# B&R Automation Studio project Palletizer (part 2)

#### Crane.st - Cyclic code
```iecst
PROGRAM _CYCLIC

	CASE State OF

		C_StopSequence:

			StartCrane			:= FALSE;
			GantryCrane.Command	:= EMERGENCY_STOP_REQUEST;
			BoxCrane.Command	:= EMERGENCY_STOP_REQUEST;
			State				:= C_StopDONE;

		C_StopDONE:

			IF (GantryCranePositionReached AND BoxCranePositionReached) THEN
				GantryCrane.Command	 := IDLE;
				BoxCrane.Command	 := IDLE;
				Crane_EmergencyStop  := FALSE;
				Crane_ImmediateStop  := FALSE;
				Crane_OnPhaseStop	 := FALSE;
				StopRequest			 := TRUE;
				State				 := C_WaitStart;
			END_IF;

		C_ResetConfig:

			IF NOT Crane_ResetConfig THEN
				State	:= C_WaitStart;
			END_IF;

			IF (GantryCranePositionReached AND BoxCranePositionReached AND NOT SlideRail_disable_request
				AND NOT PusherZ_enable_request AND NOT PusherX_enable_request AND NOT Vacuum_disable_request
				AND NOT Cartboard_disable_request) THEN

				GantryCrane.Command	:= IDLE;
				BoxCrane.Command	:= IDLE;

				FOR i := 0 TO 9 DO
					GD_StatusRequest[i]	:= FALSE;
				END_FOR;

				Crane_ResetConfig := FALSE;
				State			  := C_WaitStart;

			END_IF;

		C_RestoreConfig1:

			GantryCrane.Command	:= IDLE;
			BoxCrane.Command	:= IDLE;

			FOR i := 0 TO 9 DO
				IF GD_StatusRequest[i] THEN
					CASE i OF
						0:	Vacuum_enable_request	  := TRUE;
						1:	Vacuum_disable_request	  := TRUE;
						2:	Cartboard_enable_request  := TRUE;
						3:	Cartboard_disable_request := TRUE;
						4:	SlideRail_enable_request  := TRUE;
						5:	SlideRail_disable_request := TRUE;
						6:	PusherZ_enable_request	  := TRUE;
						7:	PusherZ_disable_request	  := TRUE;
						8:	PusherX_enable_request	  := TRUE;
						9:	PusherX_disable_request	  := TRUE;
					END_CASE;
				END_IF;
			END_FOR;

			Enable_Disable_Counter	:= 70;
			State					:= C_RestoreConfig2;

		C_RestoreConfig2:

			FOR i := 0 TO 9 DO
				IF GD_StatusRequest[i] THEN
					CASE i OF

						0:  IF NOT Vacuum_enable_request THEN
								GD_StatusRequest[i]	:= FALSE;
							END_IF;

						1:  IF NOT Vacuum_disable_request THEN
								GD_StatusRequest[i]	:= FALSE;
							END_IF;

						2:  IF NOT Cartboard_enable_request THEN
								GD_StatusRequest[i]	:= FALSE;
							END_IF

						3:  IF NOT Cartboard_disable_request THEN
								GD_StatusRequest[i]	:= FALSE;
							END_IF;

						4:	IF NOT SlideRail_enable_request THEN
								GD_StatusRequest[i]	:= FALSE;
							END_IF;

						5:  IF NOT SlideRail_disable_request THEN
								GD_StatusRequest[i]	:= FALSE;
							END_IF;

						6:  IF NOT PusherZ_enable_request THEN
								GD_StatusRequest[i]	:= FALSE;
							END_IF;

						7:  IF NOT PusherZ_disable_request THEN
								GD_StatusRequest[i]	:= FALSE;
							END_IF;

						8:  IF NOT PusherX_enable_request THEN
								GD_StatusRequest[i]	:= FALSE;
							END_IF;

						9:  IF NOT PusherX_disable_request THEN
								GD_StatusRequest[i]	:= FALSE;
							END_IF;

					END_CASE;
				END_IF;
			END_FOR;

			Enable_Disable_Counter	:= Enable_Disable_Counter - 1;

			IF Enable_Disable_Counter = 0 THEN

				IF CheckPosition[0] THEN
					GantryCraneSetPoint	:= OldPosition[0];
					GantryCrane.Command	:= CHANGE_POSITION;
				END_IF;

				IF CheckPosition[1] THEN
					BoxCraneSetPoint	:= OldPosition[1];
					BoxCrane.Command	:= CHANGE_POSITION;
				END_IF;

				State	:= C_RestoreConfig3;
			END_IF;

		C_RestoreConfig3:

			IF (GantryCranePositionReached AND CheckPosition[0]) THEN
				GantryCranePositionRestored	:= TRUE;
				GantryCrane.Command			:= IDLE;
			END_IF;

			IF (BoxCranePositionReached AND CheckPosition[1]) THEN
				BoxCranePositionRestored := TRUE;
				BoxCrane.Command		 := IDLE;
			END_IF;

			IF (NOT CheckPosition[0] OR GantryCranePositionRestored) AND (NOT CheckPosition[1] OR BoxCranePositionRestored) THEN
				StopRequest	   := FALSE;
				Crane_Restart  := FALSE;
				State		   := OldState;
			END_IF;

		C_WaitStart:

			IF Crane_Restart THEN
	  			State := C_RestoreConfig1;
			END_IF;

			IF Crane_ResetConfig THEN
				CraneCartboardCounter	  := 28;
				CraneReady				  := FALSE;
				HoldBoxes				  := FALSE;
				LoadBoxesOnPallet		  := FALSE;
				BoxesOnPallet			  := FALSE;
				SlideRail_disable_request := TRUE;
				PusherZ_enable_request	  := TRUE; (* pusher down *)
				PusherX_enable_request	  := TRUE; (* pusher forward *)
				Vacuum_disable_request	  := TRUE;
				Cartboard_disable_request := TRUE;
				GantryCraneSetPoint		  := 0;
				GantryCrane.Command	      := CHANGE_POSITION;
				BoxCraneSetPoint	      := 0;
				BoxCrane.Command	      := CHANGE_POSITION;
				State	                  := C_ResetConfig;
			END_IF;

			IF (StartCrane AND NOT Crane_ResetConfig AND NOT Crane_Restart) THEN
				GantryCraneSetPoint	 := 0;
				GantryCrane.Command	 := CHANGE_POSITION;
				State				 := C_WaitGantryCraneStartPosition;
			END_IF;

			IF Crane_EmergencyStop THEN
				State	:= C_StopSequence;
			END_IF;

			IF Crane_ImmediateStop AND NOT StopRequest THEN
				OldState := State;
				State	 := C_StopSequence;
			END_IF;

			IF Crane_ImmediateStop AND StopRequest THEN
				State	:= C_StopSequence;
			END_IF;

		C_WaitGantryCraneStartPosition:

			IF (GantryCranePositionReached OR GantryCranePositionRestored) THEN
				CheckPosition[0]			:= FALSE;
				GantryCranePositionRestored	:= FALSE;
				GantryCrane.Command			:= IDLE;
				BoxCraneSetPoint			:= -0.195;
				BoxCrane.Command			:= CHANGE_POSITION;
				State						:= C_WaitCartboardLoadPosition;
			END_IF;

			IF Crane_EmergencyStop THEN
				State	:= C_StopSequence;
			END_IF;

			IF Crane_ImmediateStop THEN
				CheckPosition[0] := TRUE;
				OldPosition[0]	 := 0;  (* old Gantry Position *)
				OldState		 := State;
				State			 := C_StopSequence;
			END_IF;

		C_WaitCartboardLoadPosition:

			IF (BoxCranePositionReached OR BoxCranePositionRestored) THEN
				CheckPosition[1]		 := FALSE;
				BoxCranePositionRestored := FALSE;
				BoxCrane.Command		 := IDLE;
				Vacuum_enable_request	 := TRUE;
				Cartboard_enable_request := TRUE;
				State					 := C_WaitCartboardLoad;
			END_IF;

			IF Crane_EmergencyStop THEN
				State	:= C_StopSequence;
			END_IF;

			IF Crane_ImmediateStop THEN
				CheckPosition[1] := TRUE;
				OldPosition[1]	 := -0.195;  (* old Box Position *)
				OldState		 := State;
				State			 := C_StopSequence;
			END_IF;

		C_WaitCartboardLoad:

			IF (NOT Vacuum_enable_request AND NOT Cartboard_enable_request) THEN
				BoxCraneSetPoint	:= 0;
				BoxCrane.Command	:= CHANGE_POSITION;
	  			State				:= C_WaitBoxCraneStartPosition;
			END_IF;

			IF Crane_EmergencyStop THEN
				State := C_StopSequence;
			END_IF;

			IF Crane_ImmediateStop THEN
				GD_StatusRequest[0] := TRUE; (* vacuumEN *)
				GD_StatusRequest[2] := TRUE; (* cartboardEN *)
				OldState		    := State;
				State				:= C_StopSequence;
			END_IF;

		C_WaitBoxCraneStartPosition:

			IF (BoxCranePositionReached OR BoxCranePositionRestored)THEN
				CheckPosition[1]		 := FALSE;
				BoxCranePositionRestored := FALSE;
				BoxCrane.Command		 := IDLE;
				PusherZ_enable_request 	 := TRUE; (* pusher down *)
				State					 := C_WaitPusherZStartDown;
			END_IF;

			IF Crane_EmergencyStop THEN
				State	:= C_StopSequence;
			END_IF;

			IF Crane_ImmediateStop THEN
				CheckPosition[1] := TRUE;
				OldPosition[1]	 := 0;  (* old Box Position *)
				OldState		 := State;
				State			 := C_StopSequence;
			END_IF;

		C_WaitPusherZStartDown:

			IF NOT PusherZ_enable_request THEN
				PusherX_enable_request := TRUE; (* pusher forward *)
				State				   := C_WaitPusherXStartFwd;
			END_IF;

			IF Crane_EmergencyStop THEN
				State	:= C_StopSequence;
			END_IF;

			IF Crane_ImmediateStop THEN
				GD_StatusRequest[6] := TRUE; (* PusherZ_EN *)
				OldState			:= State;
				State				:= C_StopSequence;
			END_IF;

		C_WaitPusherXStartFwd:

			IF NOT PusherX_enable_request THEN
				Cartboard_disable_request := TRUE;
				State					  := C_LockCartboard;
			END_IF;

			IF Crane_EmergencyStop THEN
				State	:= C_StopSequence;
			END_IF;

			IF Crane_ImmediateStop THEN
				GD_StatusRequest[8] := TRUE; (* PusherX_EN *)
				OldState		    := State;
				State				:= C_StopSequence;
			END_IF;

		C_LockCartboard:

			IF NOT Cartboard_disable_request THEN
				CraneCartboardCounter	:= CraneCartboardCounter - 1;
				CraneReady				:= TRUE;
				State					:= C_WaitBoxes;
			END_IF;

			IF Crane_EmergencyStop THEN
				State	:= C_StopSequence;
			END_IF;

			IF Crane_ImmediateStop THEN
				GD_StatusRequest[3] := TRUE; (* CartboardDIS *)
				OldState			:= State;
				State				:= C_StopSequence;
			END_IF;

		C_WaitBoxes:

			IF HoldBoxes THEN
				SlideRail_enable_request := TRUE;
				State					 := C_WaitSlideRailHold;
			END_IF;

			IF Crane_EmergencyStop THEN
				State	:= C_StopSequence;
			END_IF;

			IF Crane_ImmediateStop OR Crane_OnPhaseStop THEN
				OldState := State;
				State	 := C_StopSequence;
			END_IF;

		C_WaitSlideRailHold:

			IF NOT SlideRail_enable_request THEN
				PusherZ_disable_request	:= TRUE; (* pusher up *)
				State					:= C_WaitPusherZPushUp;
			END_IF;

			IF Crane_EmergencyStop THEN
				State	:= C_StopSequence;
			END_IF;

			IF Crane_ImmediateStop THEN
				GD_StatusRequest[4] := TRUE; (* SlideRailEN *)
				OldState			:= State;
				State				:= C_StopSequence;
			END_IF;

		C_WaitPusherZPushUp:

			IF NOT PusherZ_disable_request THEN
				PusherX_disable_request	:= TRUE; (* pusher backward *)
				State					:= C_WaitPusherXPushBwd;
			END_IF;

			IF Crane_EmergencyStop THEN
				State	:= C_StopSequence;
			END_IF;

			IF Crane_ImmediateStop THEN
				GD_StatusRequest[7] := TRUE; (* PusherZ_DIS *)
				OldState			:= State;
				State				:= C_StopSequence;
			END_IF;

		C_WaitPusherXPushBwd:

			IF NOT PusherX_disable_request THEN
				PusherZ_enable_request := TRUE; (* pusher down *)
	  			State				   := C_Idle;
			END_IF;

			IF Crane_EmergencyStop THEN
				State	:= C_StopSequence;
			END_IF;

			IF Crane_ImmediateStop THEN
				GD_StatusRequest[9] := TRUE; (* PusherX_DIS *)
				OldState			:= State;
				State				:= C_StopSequence;
			END_IF;

		C_Idle:

			IF (LoadBoxesOnPallet AND NOT PusherZ_enable_request) THEN
	  			State	:= C_WaitPusherZPushDown;
			END_IF;

			IF Crane_EmergencyStop THEN
				State	:= C_StopSequence;
			END_IF;

			IF Crane_ImmediateStop THEN
				GD_StatusRequest[6] := TRUE; (* PusherZ_EN *)
				OldState		    := State;
				State				:= C_StopSequence;
			END_IF;

		C_WaitPusherZPushDown:

			IF NOT SecondLayer THEN
				BoxCraneSetPoint := -0.2;
				BoxCrane.Command := CHANGE_POSITION;
				State			 := C_WaitBoxCraneCartboardPos;
			END_IF;

			IF SecondLayer THEN
				BoxCraneSetPoint := 0.01;
				BoxCrane.Command := CHANGE_POSITION;
				State			 := C_WaitBoxCraneCartboardPos;
			END_IF;

			IF Crane_EmergencyStop THEN
				State	:= C_StopSequence;
			END_IF;

			IF Crane_ImmediateStop THEN
				OldState := State;
				State	 := C_StopSequence;
			END_IF;

		C_WaitBoxCraneCartboardPos:

			IF (BoxCranePositionReached OR BoxCranePositionRestored) THEN
				CheckPosition[1]		 := FALSE;
				BoxCranePositionRestored := FALSE;
				BoxCrane.Command		 := IDLE;
				GantryCraneSetPoint		 := -1.11;
				GantryCrane.Command	     := CHANGE_POSITION;
				State					 := C_WaitGantryCraneCartboardPos;
			END_IF;

			IF Crane_EmergencyStop THEN
				State	:= C_StopSequence;
			END_IF;

			IF Crane_ImmediateStop THEN
				CheckPosition[1] := TRUE;

				IF NOT SecondLayer THEN
	  				OldPosition[1] := -0.2;
				END_IF;
				IF SecondLayer THEN
					OldPosition[1] := 0.01;
				END_IF;

				OldState := State;
				State	 := C_StopSequence;
			END_IF;

		C_WaitGantryCraneCartboardPos:

			IF (GantryCranePositionReached OR GantryCranePositionRestored) THEN
				CheckPosition[0]			:= FALSE;
				GantryCranePositionRestored	:= FALSE;
				GantryCrane.Command			:= IDLE;
				Vacuum_disable_request		:= TRUE;
				State						:= C_CartboardPosOk;
			END_IF;

			IF Crane_EmergencyStop THEN
				State	:= C_StopSequence;
			END_IF;

			IF Crane_ImmediateStop THEN
				CheckPosition[0] := TRUE;
				OldPosition[0]	 := -1.11;
				OldState		 := State;
				State			 := C_StopSequence;
			END_IF;

		C_CartboardPosOk:

			IF NOT Vacuum_disable_request THEN
				GantryCraneSetPoint	:= -1.3;
				GantryCrane.Command	:= CHANGE_POSITION;
				State				:= C_BoxesPosOk;
			END_IF;

			IF Crane_EmergencyStop THEN
				State	:= C_StopSequence;
			END_IF;

			IF Crane_ImmediateStop THEN
				GD_StatusRequest[1] := TRUE; (* Vacuum_DIS *)
				OldState			:= State;
				State				:= C_StopSequence;
			END_IF;

		C_BoxesPosOk:

			IF (GantryCranePositionReached OR GantryCranePositionRestored) THEN
				CheckPosition[0]			:= FALSE;
				GantryCranePositionRestored	:= FALSE;
				GantryCrane.Command			:= IDLE;
				SlideRail_disable_request	:= TRUE;
				State						:= C_OpenSlideRail;
			END_IF;

			IF Crane_EmergencyStop THEN
				State	:= C_StopSequence;
			END_IF;

			IF Crane_ImmediateStop THEN
				CheckPosition[0] := TRUE;
				OldPosition[0]	 := -1.3;
				OldState		 := State;
				State			 := C_StopSequence;
			END_IF;

		C_OpenSlideRail:

			IF NOT SlideRail_disable_request THEN
				PusherX_enable_request	:= TRUE;
				GantryCraneSetPoint		:= 0;
				GantryCrane.Command		:= CHANGE_POSITION;
				State					:= C_PusherFwd;
			END_IF;

			IF Crane_EmergencyStop THEN
				State	:= C_StopSequence;
			END_IF;

			IF Crane_ImmediateStop THEN
				GD_StatusRequest[5] := TRUE;  (* SlideRailDIS *)
				OldState			:= State;
				State				:= C_StopSequence;
			END_IF;

		C_PusherFwd:

			IF (NOT PusherX_enable_request AND (GantryCranePositionReached OR GantryCranePositionRestored)) THEN
				CheckPosition[0]			:= FALSE;
				GantryCranePositionRestored	:= FALSE;
				GantryCrane.Command			:= IDLE;
				BoxesOnPallet				:= TRUE;
				State						:= C_WaitStart;
			END_IF;

			IF Crane_EmergencyStop THEN
				State	:= C_StopSequence;
			END_IF;

			IF Crane_ImmediateStop THEN
				GD_StatusRequest[8] := TRUE; (* PusherX_EN *)
				CheckPosition[0]	:= TRUE;
				OldPosition[0]		:= 0;
				OldState			:= State;
				State				:= C_StopSequence;
			END_IF;

	END_CASE;

	(*** Generic Devices ***)

	Vacuum.DeviceOperation 			:= OperationType;
	Vacuum.DeviceClock 	   			:= TRUE;
	Vacuum.DeviceDiagnosticsEnabled := TRUE;
	Vacuum.DeviceEnablePreset 		:= FALSE;
	Vacuum.DeviceEnabledSensor 		:= Crane_Vacuum;	(* enable feedback *)
	Vacuum.DeviceEnableTime 		:= VacuumEnableTime;
	Vacuum.DeviceDisableTime 		:= VacuumDisableTime;
	Vacuum.DeviceType 				:= DEVICE_WITH_ENABLE_FEEDBACK OR DEVICE_WITH_SINGLE_ACTUATION;
	Vacuum	 ( DeviceEnableRequest  := Vacuum_enable_request,
		       DeviceDisableRequest := Vacuum_disable_request );
	Crane_VacuumGrip	 			:= Vacuum.EnableDevice;	(* single actuation *)
	act_VacuumFault 				:= SIMVacuumFault;

	Cartboard.DeviceOperation 		   := OperationType;
	Cartboard.DeviceClock 			   := TRUE;
	Cartboard.DeviceDiagnosticsEnabled := TRUE;
	Cartboard.DeviceEnablePreset 	   := FALSE;
	Cartboard.DeviceEnableTime 		   := CartboardEnableTime;
	Cartboard.DeviceDisableTime 	   := CartboardDisableTime;
	Cartboard.DeviceType 			   := DEVICE_WITHOUT_FEEDBACK OR DEVICE_WITH_SINGLE_ACTUATION;
	Cartboard	( DeviceEnableRequest  := Cartboard_enable_request,
				  DeviceDisableRequest := Cartboard_disable_request );
	Crane_CartboardTrig 			   := Cartboard.EnableDevice;	(* single actuation *)
	act_CartboardFault				   := SIMCartboardFault;

	SlideRail.DeviceOperation 		   := OperationType;
	SlideRail.DeviceClock 			   := TRUE;
	SlideRail.DeviceDiagnosticsEnabled := TRUE;
	SlideRail.DeviceEnablePreset 	   := FALSE;
	SlideRail.DeviceEnableTime 		   := SlideRailEnableTime;
	SlideRail.DeviceDisableTime 	   := SlideRailDisableTime;
	SlideRail.DeviceType 			   := DEVICE_WITHOUT_FEEDBACK OR DEVICE_WITH_SINGLE_ACTUATION;
	SlideRail	( DeviceEnableRequest  := SlideRail_enable_request,
				  DeviceDisableRequest := SlideRail_disable_request );
	Crane_SlideRail_EN 			   	   := SlideRail.EnableDevice;  (* single actuation *)
	act_SlideRailFault				   := SIMSlideRailFault;

	PusherZ.DeviceOperation 		 := OperationType;
	PusherZ.DeviceClock 			 := TRUE;
	PusherZ.DeviceDiagnosticsEnabled := TRUE;
	PusherZ.DeviceEnablePreset 		 := FALSE;
	PusherZ.DeviceEnableTime 		 := PusherZEnableTime;
	PusherZ.DeviceDisableTime 		 := PusherZDisableTime;
	PusherZ.DeviceType 				 := DEVICE_WITHOUT_FEEDBACK OR DEVICE_WITH_SINGLE_ACTUATION;
	PusherZ	  ( DeviceEnableRequest  := PusherZ_enable_request,
				DeviceDisableRequest := PusherZ_disable_request );
	Crane_PusherZ_EN 				 := PusherZ.EnableDevice;  (* single actuation *)
	act_PusherZFault				 := SIMPusherZFault;

	PusherX.DeviceOperation 		 := OperationType;
	PusherX.DeviceClock 			 := TRUE;
	PusherX.DeviceDiagnosticsEnabled := TRUE;
	PusherX.DeviceEnablePreset 		 := FALSE;
	PusherX.DeviceEnableTime 		 := PusherXEnableTime;
	PusherX.DeviceDisableTime 		 := PusherXDisableTime;
	PusherX.DeviceType 				 := DEVICE_WITHOUT_FEEDBACK OR DEVICE_WITH_SINGLE_ACTUATION;
	PusherX    ( DeviceEnableRequest := PusherX_enable_request,
				DeviceDisableRequest := PusherX_disable_request );
	Crane_PusherX_EN 				 := PusherX.EnableDevice;  (* single actuation *)
	act_PusherXFault				 := SIMPusherXFault;

	(*** Generic Axes ***)

	GantryCrane.NewSetPoint		:= GantryCraneSetPoint;
	GantryCrane.ActualPosition	:= Crane_Gantry_Axis;
	GantryCrane.TGT_SENSOR		:= TRUE;
	Crane_Gantry_Axis_TgtPos	:= GantryCrane.TargetPosition;
	GantryCranePositionReached	:= GantryCrane.InPosition;
	GantryCrane.DeviceTimer		:= 400;
	act_GantryCraneFault		:= SIMGantryCraneFault;
	GantryCrane();

	BoxCrane.NewSetPoint	:= BoxCraneSetPoint;
	BoxCrane.ActualPosition	:= Crane_Box_Axis;
	BoxCrane.TGT_SENSOR		:= TRUE;
	Crane_Box_Axis_TgtPos	:=	BoxCrane.TargetPosition;
	BoxCranePositionReached	:= BoxCrane.InPosition;
	BoxCrane.DeviceTimer	:= 400;
	act_BoxCraneFault		:= SIMBoxCraneFault;
	BoxCrane();

END_PROGRAM
```

#### Types.typ - Local data types
```iecst
TYPE
	CraneState :
		(
		C_StopSequence := 1,
		C_StopDONE := 2,
		C_ResetConfig := 3,
		C_RestoreConfig1 := 4,
		C_RestoreConfig2 := 5,
		C_RestoreConfig3 := 6,
		C_WaitStart := 7,
		C_WaitGantryCraneStartPosition := 8,
		C_WaitCartboardLoadPosition := 9,
		C_WaitCartboardLoad := 10,
		C_WaitBoxCraneStartPosition := 11,
		C_WaitPusherZStartDown := 12,
		C_WaitPusherXStartFwd := 13,
		C_LockCartboard := 14,
		C_WaitBoxes := 15,
		C_WaitSlideRailHold := 16,
		C_WaitPusherZPushUp := 17,
		C_WaitPusherXPushBwd := 18,
		C_Idle := 19,
		C_WaitPusherZPushDown := 20,
		C_WaitBoxCraneCartboardPos := 21,
		C_WaitGantryCraneCartboardPos := 22,
		C_CartboardPosOk := 23,
		C_BoxesPosOk := 24,
		C_OpenSlideRail := 25,
		C_PusherFwd := 26
		);
END_TYPE
```

#### Variables.var - Local variables
```iecst
VAR
	GantryCranePositionRestored : BOOL := FALSE;
END_VAR
(*Vacuum*)
VAR
	BoxCranePositionReached : BOOL;
	GantryCranePositionReached : BOOL;
	StopRequest : BOOL := FALSE;
	BoxCranePositionRestored : BOOL := FALSE;
	CheckPosition : ARRAY[0..1] OF BOOL := [2(FALSE)];
END_VAR
(*Faults*)
VAR
	GD_StatusRequest : ARRAY[0..9] OF BOOL := [10(FALSE)];
	OldState : CraneState;
	State : CraneState := C_WaitStart;
END_VAR
(*GantryCrane*)
VAR
	GantryCrane : GenericAxis;
END_VAR
(*BoxCrane*)
VAR
	BoxCrane : GenericAxis;
END_VAR
(*SlideRail*)
VAR
	SlideRail : GenericDevice;
END_VAR
(*PusherX*)
VAR
	PusherX : GenericDevice;
END_VAR
(*PusherZ*)
VAR
	PusherZ : GenericDevice;
END_VAR
(*Cartboard*)
VAR
	Cartboard : GenericDevice;
	Vacuum : GenericDevice;
	Enable_Disable_Counter : INT;
	VacuumDisableTime : INT := 80;
	PusherZDisableTime : INT := 60;
	CartboardDisableTime : INT := 60;
	VacuumEnableTime : INT := 80;
	SlideRailEnableTime : INT := 60;
	SlideRailDisableTime : INT := 60;
	PusherXDisableTime : INT := 60;
	PusherZEnableTime : INT := 60;
	CartboardEnableTime : INT := 60;
	PusherXEnableTime : INT := 60;
	i : INT := 0;
	GantryCraneSetPoint : REAL;
	BoxCraneSetPoint : REAL;
	OldPosition : ARRAY[0..1] OF REAL;
END_VAR
```

### Program Logical/PalletHandler (IEC)

#### Pallet.st - Cyclic code
```iecst
PROGRAM _CYCLIC

	CASE State OF

		P_StopSequence:

			StartPallet				    	:= FALSE;
			PalletConveyor1_disable_request	:= TRUE;
			PalletLifter.Command			:= EMERGENCY_STOP_REQUEST;
			PalletConveyor2.Command			:= EMERGENCY_STOP_REQUEST;
			State							:= P_StopDONE;

		P_StopDONE:

			IF (NOT PalletConveyor1_disable_request AND PalletLifterPositionReached AND PalletConveyor2VelocityReached) THEN
				PalletLifter.Command	:= IDLE;
				PalletConveyor2.Command	:= IDLE;
				Pallet_EmergencyStop	:= FALSE;
				Pallet_ImmediateStop	:= FALSE;
				Pallet_OnPhaseStop		:= FALSE;
				StopRequest				:= TRUE;
				State					:= P_WaitStart;
			END_IF;

		P_ResetConfig1:

			IF NOT Pallet_ResetConfig THEN
				State	:= P_WaitStart;
			END_IF;

			IF PalletLifterPositionReached THEN
				PalletLifter.Command	   := IDLE;
				PalletFork_disable_request := TRUE; (* fork closed *)
				State					   := P_ResetConfig2;
			END_IF;

		P_ResetConfig2:

			IF NOT PalletFork_disable_request THEN
				PalletLifterSetPoint	:= 0; (* idle position *)
				PalletLifter.Command	:= CHANGE_POSITION;
				State					:= P_ResetConfig3;
			END_IF;

		P_ResetConfig3:

			IF PalletLifterPositionReached THEN
				PalletLifter.Command := IDLE;

				FOR i := 0 TO 3 DO
					GD_StatusRequest[i] := FALSE;
				END_FOR;

				Pallet_ResetConfig := FALSE;
				State			   := P_WaitStart;
			END_IF;

		P_RestoreConfig1:

			PalletLifter.Command	:= IDLE;
			PalletConveyor2.Command	:= IDLE;

			FOR i := 0 TO 3 DO
				IF GD_StatusRequest[i] THEN
					CASE i OF
						0:	PalletFork_enable_request		:= TRUE;
						1:	PalletFork_disable_request		:= TRUE;
						2:	PalletConveyor1_enable_request	:= TRUE;
						3:	PalletConveyor1_disable_request	:= TRUE;
					END_CASE;
				END_IF;
			END_FOR;

			Enable_Disable_Counter	:= 70;
			State					:= P_RestoreConfig2;

		P_RestoreConfig2:

			FOR i := 0 TO 3 DO
				IF GD_StatusRequest[i] THEN
					CASE i OF
						0: IF NOT PalletFork_enable_request THEN
								GD_StatusRequest[i]	:= FALSE;
							END_IF;

						1: IF NOT PalletFork_disable_request THEN
								GD_StatusRequest[i]	:= FALSE;
							END_IF;

						2: IF NOT PalletConveyor1_enable_request THEN
								GD_StatusRequest[i]	:= FALSE;
							END_IF;

						3: IF NOT PalletConveyor1_disable_request THEN
								GD_StatusRequest[i]	:= FALSE;
							END_IF;
					END_CASE;
				END_IF;
			END_FOR;

			Enable_Disable_Counter	:= Enable_Disable_Counter - 1;

			IF Enable_Disable_Counter = 0 THEN
				IF CheckPosition THEN
					PalletLifterSetPoint	:= OldPosition;
					PalletLifter.Command	:= CHANGE_POSITION;
				END_IF;

				IF CheckVelocity THEN
					PalletConveyor2SetPoint	:= OldVelocity;
					PalletConveyor2.Command	:= CHANGE_VELOCITY;
				END_IF;

				State	:= P_RestoreConfig3;
			END_IF;

		P_RestoreConfig3:

			IF (PalletLifterPositionReached AND CheckPosition) THEN
				PalletLifterPositionRestored := TRUE;
				PalletLifter.Command		 := IDLE;
			END_IF;

			IF (PalletConveyor2VelocityReached AND CheckVelocity) THEN
				PalletConveyor2VelocityRestored	:= TRUE;
				PalletConveyor2.Command			:= IDLE;
			END_IF;

			IF (NOT CheckPosition OR PalletLifterPositionReached) AND (NOT CheckVelocity OR PalletConveyor2VelocityReached) THEN
				StopRequest		:= FALSE;
				Pallet_Restart	:= FALSE;
				State			:= OldState;
			END_IF;

		P_WaitStart:

			IF Pallet_Restart THEN
				State	:= P_RestoreConfig1;
			END_IF;

			IF Pallet_ResetConfig THEN
				PalletCounter	:= 5;
				PalletReady		:= FALSE;
				PalletExit_EN	:= FALSE;
				PalletExit_DONE	:= FALSE;

				IF PalletFork.DeviceDisabled THEN (* fork closed *)
					PalletLifterSetPoint := 0; (* idle position *)
					PalletLifter.Command := CHANGE_POSITION;
					State				 := P_ResetConfig3;
				ELSE (* fork opened *)
					PalletLifterSetPoint := -0.258;
					PalletLifter.Command := CHANGE_POSITION;
					State				 := P_ResetConfig1;
				END_IF;

			END_IF;

			IF (StartPallet AND NOT Pallet_ResetConfig AND NOT Pallet_Restart) THEN
				PalletLifterSetPoint := -0.258;
				PalletLifter.Command := CHANGE_POSITION;
				State				 := P_WaitLifterDown;
			END_IF;

			IF Pallet_EmergencyStop THEN
				State := P_StopSequence;
			END_IF;

			IF Pallet_ImmediateStop AND NOT StopRequest THEN
				IF PalletOnConveyor2 THEN
					CheckVelocity		:= TRUE;
					OldVelocity			:= 0.5;  (* old conveyor 2 velocity *) //0.3
					PalletOnConveyor2	:= FALSE;
				END_IF;

				OldState	:= State;
				State		:= P_StopSequence;
			END_IF;

			IF Pallet_ImmediateStop AND StopRequest THEN
				State	:= P_StopSequence;
			END_IF;

		P_WaitLifterDown:

			IF (PalletLifterPositionReached OR PalletLifterPositionRestored) THEN
				CheckPosition				 := FALSE;
				PalletLifterPositionRestored := FALSE;
				PalletLifter.Command		 := IDLE;
				PalletFork_enable_request	 := TRUE;
				State						 := P_ForkOpen;
			END_IF;

			IF Pallet_EmergencyStop THEN
				State := P_StopSequence;
			END_IF;

			IF Pallet_ImmediateStop OR Pallet_OnPhaseStop THEN
				IF PalletOnConveyor2 THEN
					CheckVelocity	  := TRUE;
					OldVelocity		  := 0.5; (* old conveyor 2 velocity *) //0.3
					PalletOnConveyor2 := FALSE;
				END_IF;

				CheckPosition	:= TRUE;
				OldPosition		:= -0.258; (* old pallet lifter position *)
				OldState		:= State;
				State			:= P_StopSequence;
			END_IF;

		P_ForkOpen:

			IF NOT PalletFork_enable_request THEN
				PalletLifterSetPoint := -0.12;
				PalletLifter.Command := CHANGE_POSITION;
				State				 := P_WaitLifterUp;
			END_IF;

			IF Pallet_EmergencyStop THEN
				State := P_StopSequence;
			END_IF;

			IF Pallet_ImmediateStop THEN
				IF PalletOnConveyor2 THEN
					CheckVelocity 	  := TRUE;
					OldVelocity	  	  := 0.5; (* old conveyor 2 velocity *) //0.3
					PalletOnConveyor2 := FALSE;
				END_IF;

				GD_StatusRequest[0] := TRUE; (* pallet fork EN *)
				OldState			:= State;
				State				:= P_StopSequence;
			END_IF;

		P_WaitLifterUp:

			IF (PalletLifterPositionReached OR PalletLifterPositionRestored) THEN
				CheckPosition				 := FALSE;
				PalletLifterPositionRestored := FALSE;
				PalletLifter.Command		 := IDLE;
				PalletFork_disable_request	 := TRUE;
				State						 := P_ForkClose;
			END_IF;

			IF Pallet_EmergencyStop THEN
				State := P_StopSequence;
			END_IF;

			IF Pallet_ImmediateStop THEN
				CheckPosition := TRUE;
				OldPosition	  := -0.12; (* old pallet lifter position *)
				OldState	  := State;
				State	      := P_StopSequence;
			END_IF;

		P_ForkClose:

			IF NOT PalletFork_disable_request  THEN
				PalletLifterSetPoint := 0.0;
				PalletLifter.Command := CHANGE_POSITION;
				State				 := P_WaitLifterIdle;
			END_IF;

			IF Pallet_EmergencyStop THEN
				State := P_StopSequence;
			END_IF;

			IF Pallet_ImmediateStop THEN
				GD_StatusRequest[1] := TRUE; (* pallet fork DIS *)
				OldState			:= State;
				State				:= P_StopSequence;
			END_IF;

		P_WaitLifterIdle:

			IF (PalletLifterPositionReached OR PalletLifterPositionRestored) THEN
				CheckPosition				 	:= FALSE;
				PalletLifterPositionRestored 	:= FALSE;
				PalletLifter.Command		 	:= IDLE;
				PalletCounter				 	:= PalletCounter -1;
				PalletConveyor1_enable_request	:= TRUE;
				State							:= P_WaitConveyor1;
			END_IF;

			IF Pallet_EmergencyStop THEN
				State := P_StopSequence;
			END_IF;

			IF Pallet_ImmediateStop THEN
				CheckPosition	:= TRUE;
				OldPosition		:= 0.0; (* old pallet lifter position *)
				OldState		:= State;
				State			:= P_StopSequence;
			END_IF;

		P_WaitConveyor1:

			IF NOT PalletConveyor1_enable_request THEN
				PalletConveyor2SetPoint	:= 0.5;
				PalletConveyor2.Command	:= CHANGE_VELOCITY;
				State					:= P_WaitConveyor2;
			END_IF;

			IF Pallet_EmergencyStop THEN
				State := P_StopSequence;
			END_IF;

			IF Pallet_ImmediateStop THEN
				GD_StatusRequest[2] := TRUE; (* pallet conveyor 1 EN *)
				OldState			:= State;
				State				:= P_StopSequence;
			END_IF;

		P_WaitConveyor2:

			IF (PalletConveyor2VelocityReached OR PalletConveyor2VelocityRestored) THEN
				CheckVelocity					:= FALSE;
				PalletConveyor2VelocityRestored	:= FALSE;
				PalletConveyor2.Command			:= IDLE;
				State							:= P_WaitLightBarrier2;
			END_IF;

			IF Pallet_EmergencyStop THEN
				State	:= P_StopSequence;
			END_IF;

			IF Pallet_ImmediateStop THEN
				GD_StatusRequest[2] := TRUE; (* pallet conveyor 1 EN *)
				CheckVelocity		:= TRUE;
				OldVelocity			:= 0.5;  (* old conveyor 2 velocity *)
				OldState			:= State;
				State				:= P_StopSequence;
			END_IF;

		P_WaitLightBarrier2:

			IF LightBarrier2 AND (PalletConveyor2VelocityRestored OR NOT CheckVelocity) THEN
				CheckVelocity					:= FALSE;
				PalletConveyor2VelocityRestored	:= FALSE;
				PalletConveyor1_disable_request	:= TRUE;
				State							:= P_WaitStopConveyor1;
			END_IF;

			IF Pallet_EmergencyStop THEN
				State := P_StopSequence;
			END_IF;

			IF Pallet_ImmediateStop THEN
				GD_StatusRequest[2] := TRUE; (* pallet conveyor 1 EN *)
				CheckVelocity		:= TRUE;
				OldVelocity			:= 0.5; (* old conveyor 2 velocity *)
				OldState			:= State;
				State				:= P_StopSequence;
			END_IF;

		P_WaitStopConveyor1:

			IF NOT PalletConveyor1_disable_request AND (PalletConveyor2VelocityRestored OR NOT CheckVelocity) THEN
				CheckVelocity					:= FALSE;
				PalletConveyor2VelocityRestored	:= FALSE;
				PalletConveyor2SetPoint			:= 0.1;
				PalletConveyor2.Command			:= CHANGE_VELOCITY;
				State							:= P_WaitConveyor2SlowDown;
			END_IF;

			IF Pallet_EmergencyStop THEN
				State := P_StopSequence;
			END_IF;

			IF Pallet_ImmediateStop THEN
				CheckVelocity			  := TRUE;
				OldVelocity				  := 0.5;  (* old conveyor 2 velocity *)
				GD_StatusRequest[3] 	  := TRUE; (* pallet conveyor 1 DIS *)
				OldState				  := State;
				State					  := P_StopSequence;
			END_IF;

		P_WaitConveyor2SlowDown:

			IF (PalletConveyor2VelocityReached OR PalletConveyor2VelocityRestored) THEN
				CheckVelocity					:= FALSE;
				PalletConveyor2VelocityRestored	:= FALSE;
				PalletConveyor2.Command			:= IDLE;
				State							:= P_WaitLightBarrier1;
			END_IF;

			IF Pallet_EmergencyStop THEN
				State := P_StopSequence;
			END_IF;

			IF Pallet_ImmediateStop THEN
				CheckVelocity			  := TRUE;
				OldVelocity				  := 0.1;  (* old conveyor 2 velocity *)
				GD_StatusRequest[3] 	  := TRUE; (* pallet conveyor 1 DIS *)
				OldState				  := State;
				State					  := P_StopSequence;
			END_IF;

		P_WaitLightBarrier1:

			IF LightBarrier1 AND (PalletConveyor2VelocityRestored OR NOT CheckVelocity) THEN
				CheckVelocity					:= FALSE;
				PalletConveyor2VelocityRestored	:= FALSE;
				PalletConveyor2SetPoint			:= 0.0;
				PalletConveyor2.Command			:= CHANGE_VELOCITY;
				State							:= P_WaitStopConveyor2;
			END_IF;

			IF Pallet_EmergencyStop THEN
				State := P_StopSequence;
			END_IF;

			IF Pallet_ImmediateStop THEN
				CheckVelocity := TRUE;
				OldVelocity	  := 0.1;  (* old conveyor 2 velocity *)
				OldState	  := State;
				State		  := P_StopSequence;
			END_IF;

		P_WaitStopConveyor2:

			IF (PalletConveyor2VelocityReached OR PalletConveyor2VelocityRestored) THEN
				CheckVelocity					:= FALSE;
				PalletConveyor2VelocityRestored	:= FALSE;
				PalletConveyor2.Command			:= IDLE;
				PalletReady						:= TRUE;
				State							:= P_WaitBoxes;
			END_IF;

			IF Pallet_EmergencyStop THEN
				State := P_StopSequence;
			END_IF;

			IF Pallet_ImmediateStop THEN
				CheckVelocity := TRUE;
				OldVelocity	  := 0.0; (* old conveyor 2 velocity *)
				OldState	  := State;
				State		  := P_StopSequence;
			END_IF;

		P_WaitBoxes:

			IF PalletExit_EN THEN
				PalletConveyor2SetPoint	:= 0.3;
				PalletConveyor2.Command	:= CHANGE_VELOCITY;
				State					:= P_WaitRestartConveyor2;
			END_IF;

			IF Pallet_EmergencyStop THEN
				State := P_StopSequence;
			END_IF;

			IF Pallet_ImmediateStop OR Pallet_OnPhaseStop THEN
				OldState := State;
				State	 := P_StopSequence;
			END_IF;

		P_WaitRestartConveyor2:

			IF (PalletConveyor2VelocityReached OR PalletConveyor2VelocityRestored) THEN
				CheckVelocity					:= FALSE;
				PalletConveyor2VelocityRestored	:= FALSE;
				PalletConveyor2.Command			:= IDLE;
				State							:= P_WaitNOTLightBarrier2;
			END_IF;

			IF Pallet_EmergencyStop THEN
				State	:= P_StopSequence;
			END_IF;

			IF Pallet_ImmediateStop THEN
				CheckVelocity := TRUE;
				OldVelocity	  := 0.3;  (* old conveyor 2 velocity *)
				OldState	  := State;
				State	      := P_StopSequence;
			END_IF;

		P_WaitNOTLightBarrier2:

			IF NOT LightBarrier2 AND (PalletConveyor2VelocityRestored OR NOT CheckVelocity) THEN
				CheckVelocity					:= FALSE;
				PalletConveyor2VelocityRestored	:= FALSE;
				PalletConveyor2SetPoint			:= 0.5;
				PalletConveyor2.Command			:= CHANGE_VELOCITY;
				State							:= P_WaitExitVelocity;
			END_IF;

			IF Pallet_EmergencyStop THEN
				State	:= P_StopSequence;
			END_IF;

			IF Pallet_ImmediateStop THEN
				CheckVelocity := TRUE;
				OldVelocity	  := 0.3; (* old conveyor 2 velocity *)
				OldState	  := State;
				State	      := P_StopSequence;
			END_IF;

		P_WaitExitVelocity:

			IF (PalletConveyor2VelocityReached OR PalletConveyor2VelocityRestored) THEN
				CheckVelocity					:= FALSE;
				PalletConveyor2VelocityRestored	:= FALSE;
				PalletConveyor2.Command			:= IDLE;
				PalletOnConveyor2				:= TRUE;
				PalletExit_DONE					:= TRUE;
				State							:= P_WaitStart;
			END_IF;

			IF Pallet_EmergencyStop THEN
				State	:= P_StopSequence;
			END_IF;

			IF Pallet_ImmediateStop THEN
				CheckVelocity	:= TRUE;
				OldVelocity		:= 0.5; (* old conveyor 2 velocity *)
				OldState		:= State;
				State			:= P_StopSequence;
			END_IF;

	END_CASE;

	(*** Generic Devices ***)

	PalletFork.DeviceOperation  		:= OperationType;
	PalletFork.DeviceClock 				:= TRUE;
	PalletFork.DeviceDiagnosticsEnabled := TRUE;
	PalletFork.DeviceEnablePreset 		:= FALSE;
	PalletFork.DeviceEnabledSensor 		:= Pallet_ForkFB;  (* enable feedback *)
	PalletFork.DeviceEnableTime 		:= PalletForkEnableTime;
	PalletFork.DeviceDisableTime 		:= PalletForkDisableTime;
	PalletFork.DeviceType 				:= DEVICE_WITH_ENABLE_FEEDBACK OR DEVICE_WITH_SINGLE_ACTUATION;
	PalletFork	 ( DeviceEnableRequest  := PalletFork_enable_request,
		           DeviceDisableRequest := PalletFork_disable_request );
	Pallet_Fork_EN		 				:= PalletFork.EnableDevice;  (* single actuation *)
	act_PalletForkFault 				:= SIMPalletForkFault;

	PalletConveyor1.DeviceOperation 		 := OperationType;
	PalletConveyor1.DeviceClock 			 := TRUE;
	PalletConveyor1.DeviceDiagnosticsEnabled := TRUE;
	PalletConveyor1.DeviceEnablePreset 		 := FALSE;
	PalletConveyor1.DeviceEnableTime 		 := PalletConveyor1EnableTime;
	PalletConveyor1.DeviceDisableTime 	     := PalletConveyor1DisableTime;
	PalletConveyor1.DeviceType 				 := DEVICE_WITHOUT_FEEDBACK OR DEVICE_WITH_SINGLE_ACTUATION;
	PalletConveyor1   ( DeviceEnableRequest  := PalletConveyor1_enable_request,
		                DeviceDisableRequest := PalletConveyor1_disable_request );
	Pallet_Conveyor1_Fwd 					 := PalletConveyor1.EnableDevice;	(* single actuation *)
	act_PalletConveyor1Fault				 := SIMPalletConveyor1Fault;

	(*** Generic Axes ***)

	PalletLifter.NewSetPoint	:= PalletLifterSetPoint;
	PalletLifter.ActualPosition	:= Pallet_Lifter_Axis;
	PalletLifter.TGT_SENSOR		:= TRUE;
	Pallet_Lifter_Axis_TgtPos 	:= PalletLifter.TargetPosition;
	PalletLifterPositionReached	:= PalletLifter.InPosition;
	PalletLifter.DeviceTimer	:= 400;
	act_PalletLifterFault		:= SIMPalletLifterFault;
	PalletLifter();

	PalletConveyor2.NewSetPoint		:= PalletConveyor2SetPoint;
	PalletConveyor2.ActualVelocity	:= Pallet_Conveyor2_ActVel;
	Pallet_Conveyor2_ActVel			:= PalletConveyor2.TargetVelocity;
	PalletConveyor2VelocityReached	:= PalletConveyor2.InVelocity;
	PalletConveyor2.DeviceTimer		:= 400;
	act_PalletConveyor2Fault		:= SIMPalletConveyor2Fault;
	PalletConveyor2();

END_PROGRAM
```

#### Types.typ - Local data types
```iecst
TYPE
	PalletState :
		(
		P_StopSequence := 1,
		P_StopDONE := 2,
		P_ResetConfig1 := 3,
		P_ResetConfig2 := 4,
		P_ResetConfig3 := 5,
		P_RestoreConfig1 := 6,
		P_RestoreConfig2 := 7,
		P_RestoreConfig3 := 8,
		P_WaitStart := 9,
		P_WaitLifterDown := 10,
		P_ForkOpen := 11,
		P_WaitLifterUp := 12,
		P_ForkClose := 13,
		P_WaitLifterIdle := 14,
		P_WaitConveyor1 := 15,
		P_WaitConveyor2 := 16,
		P_WaitLightBarrier2 := 17,
		P_WaitStopConveyor1 := 18,
		P_WaitConveyor2SlowDown := 19,
		P_WaitLightBarrier1 := 20,
		P_WaitStopConveyor2 := 21,
		P_WaitBoxes := 22,
		P_WaitRestartConveyor2 := 23,
		P_WaitNOTLightBarrier2 := 24,
		P_WaitExitVelocity := 25
		);
END_TYPE
```

#### Variables.var - Local variables
```iecst
VAR
	State : PalletState := P_WaitStart;
END_VAR
(*PalletFork*)
VAR
	PalletFork : GenericDevice;
	PalletForkEnableTime : INT := 80;
	PalletForkDisableTime : INT := 80;
END_VAR
(*Pallet Lifter*)
VAR
	PalletLifter : GenericAxis;
	PalletLifterPositionReached : BOOL;
	PalletLifterSetPoint : REAL;
END_VAR
(*Pallet Conveyor 1*)
VAR
	PalletConveyor1 : GenericDevice;
	PalletConveyor1EnableTime : INT := 20;
	PalletConveyor1DisableTime : INT := 20;
END_VAR
(*Pallet Conveyor 2*)
VAR
	PalletConveyor2 : GenericAxis;
	PalletConveyor2VelocityReached : BOOL;
	PalletConveyor2SetPoint : REAL;
	GD_StatusRequest : ARRAY[0..3] OF BOOL := [4(FALSE)];
	i : INT;
	Enable_Disable_Counter : INT;
	CheckPosition : BOOL := FALSE;
	OldPosition : REAL;
	CheckVelocity : BOOL := FALSE;
	OldVelocity : REAL;
	PalletLifterPositionRestored : BOOL := FALSE;
	OldState : PalletState;
	PalletConveyor2VelocityRestored : BOOL := FALSE;
	PalletOnConveyor2 : BOOL := FALSE;
	StopRequest : BOOL := FALSE;
END_VAR
```

### Program Logical/TaskManager (IEC)

#### Types.typ
```iecst
TYPE
	Main_State :
		(
		M_EmergencyStopSequence := 1,
		M_StopSequence := 2,
		M_Restart := 3,
		M_WaitStart := 4,
		M_BoxPosOk := 5,
		M_BoxOnCrane := 6,
		M_WaitForPallet := 7,
		M_BoxOnPallet := 8,
		M_PalletExit := 9
		);
END_TYPE
```

#### Variables.var
```iecst
VAR
	State : Main_State := M_WaitStart;
	RestartRequest : BOOL := FALSE;
	OldState : Main_State;
	ImmediateStopRequest : BOOL := FALSE;
	OnPhaseStopRequest : BOOL := FALSE;
	StopRequest : BOOL := FALSE;
	PalletOutput : INT := 0;
END_VAR
```

#### Main.st
```iecst
PROGRAM _CYCLIC

	CASE State OF

		// Recovery of the machine from the Emergency Stop - Every state can be sent here to recover

		M_EmergencyStopSequence:

			EnableMachine	:= FALSE;
			StartMachine	:= FALSE;
			IF (NOT EmergencyStop AND NOT Feeder_EmergencyStop AND NOT Crane_EmergencyStop AND NOT Pallet_EmergencyStop) THEN
				Feeder_ResetConfig := TRUE;
				Crane_ResetConfig  := TRUE;
				Pallet_ResetConfig := TRUE;
				RestartRequest	   := FALSE;
				State			   := M_WaitStart;
			END_IF;

		// Recovery of the machine from the Immediate Stop (caused by Faults) and the On Phase Stop - Every state can be sent here to recover

		M_StopSequence:

			EnableMachine	:= FALSE;
			StartMachine	:= FALSE;
			StopRequest		:= TRUE;
			IF (NOT ImmediateStop AND NOT Feeder_EmergencyStop AND NOT Crane_EmergencyStop AND NOT Pallet_EmergencyStop)
				AND (NOT OnPhaseStop AND NOT Feeder_OnPhaseStop AND NOT Crane_OnPhaseStop AND NOT Pallet_OnPhaseStop) THEN
				EnableMachine	:= TRUE;
				RestartRequest	:= TRUE;
				State			:= M_WaitStart;
			END_IF;

			IF EmergencyStop AND (OnPhaseStopRequest OR ImmediateStopRequest) THEN
				OnPhaseStopRequest		:= FALSE;
				ImmediateStopRequest	:= FALSE;
				Feeder_ImmediateStop	:= FALSE;
				Crane_ImmediateStop		:= FALSE;
				Pallet_ImmediateStop	:= FALSE;
				Feeder_OnPhaseStop		:= FALSE;
				Crane_OnPhaseStop		:= FALSE;
				Pallet_OnPhaseStop		:= FALSE;
				State					:= M_WaitStart;
			END_IF;

			IF ImmediateStop AND OnPhaseStopRequest THEN
				OnPhaseStopRequest		:= FALSE;
				Feeder_OnPhaseStop		:= FALSE;
				Crane_OnPhaseStop		:= FALSE;
				Pallet_OnPhaseStop		:= FALSE;
				State					:= M_WaitStart;

			END_IF;

		// Machine restarts when coming from Faults and Stops

		M_Restart:

			IF (NOT Feeder_Restart AND NOT Crane_Restart AND NOT Pallet_Restart) THEN
				StopRequest		:= FALSE;
				RestartRequest	:= FALSE;
				StartFeeder		:= TRUE;
				StartCrane		:= TRUE;
				StartPallet 	:= TRUE;
				State			:= OldState;
			END_IF;

		// Machine starting procedure

		M_WaitStart:

			// Restart machine after Stops or Faults

			IF (StartMachine AND EnableMachine AND RestartRequest) THEN
				Feeder_Restart := TRUE;
				Crane_Restart  := TRUE;
				Pallet_Restart := TRUE;
				State		   := M_Restart;
			END_IF;

			IF (NOT Feeder_ResetConfig AND NOT Crane_ResetConfig AND NOT Pallet_ResetConfig) THEN
				EnableMachine	:= TRUE;
			END_IF;

			// Nominal working condition

			IF (StartMachine AND EnableMachine AND NOT RestartRequest) THEN
				StartFeeder   := TRUE;
				StartCrane	  := TRUE;
				StartPallet   := TRUE;
				State		  := M_BoxPosOk;
			END_IF;

			IF EmergencyStop THEN
				Feeder_EmergencyStop := TRUE;
				Crane_EmergencyStop  := TRUE;
				Pallet_EmergencyStop := TRUE;
				State				 := M_EmergencyStopSequence;
			END_IF;

			IF ImmediateStop THEN
				ImmediateStopRequest := TRUE;

				IF NOT StopRequest THEN
					OldState := State;
				END_IF;

				Feeder_ImmediateStop := TRUE;
				Crane_ImmediateStop  := TRUE;
				Pallet_ImmediateStop := TRUE;
				State				 := M_StopSequence;
			END_IF;

			IF OnPhaseStop AND NOT StopRequest THEN
				OnPhaseStopRequest	:= TRUE;

				IF NOT StopRequest THEN
					OldState	:= State;
				END_IF;

				Feeder_OnPhaseStop := TRUE;
				Crane_OnPhaseStop  := TRUE;
				Pallet_OnPhaseStop := TRUE;
				State			   := M_StopSequence;
			END_IF;

		// A layer of boxes is ready to be placed on the BoxCrane

		M_BoxPosOk:

			PalletExit_DONE	:= FALSE;
			BoxesOnPallet	:= FALSE;

			IF (FeederReady AND CraneReady) THEN
				LoadBoxesOnCrane := TRUE;
				State			  := M_BoxOnCrane;
			END_IF;

			IF EmergencyStop THEN
				Feeder_EmergencyStop := TRUE;
				Crane_EmergencyStop  := TRUE;
				Pallet_EmergencyStop := TRUE;
				State				 := M_EmergencyStopSequence;
			END_IF;

			IF ImmediateStop THEN
				ImmediateStopRequest := TRUE;
				OldState			 := State;
				Feeder_ImmediateStop := TRUE;
				Crane_ImmediateStop  := TRUE;
				Pallet_ImmediateStop := TRUE;
				State				 := M_StopSequence;
			END_IF;

			IF OnPhaseStop THEN
				OnPhaseStopRequest := TRUE;
				OldState		   := State;
				Feeder_OnPhaseStop := TRUE;
				Crane_OnPhaseStop  := TRUE;
				Pallet_OnPhaseStop := TRUE;
				State			   := M_StopSequence;
			END_IF;

		// 	The layer of boxes is placed on the BoxCrane

		M_BoxOnCrane:

			IF BoxesOnCrane THEN
				FeederReady			:= FALSE;
				CraneReady			:= FALSE;
				LoadBoxesOnCrane	:= FALSE;
				HoldBoxes			:= TRUE;
				State				:= M_WaitForPallet;
			END_IF;

			IF EmergencyStop THEN
				Feeder_EmergencyStop := TRUE;
				Crane_EmergencyStop  := TRUE;
				Pallet_EmergencyStop := TRUE;
				State				 := M_EmergencyStopSequence;
			END_IF;

			IF ImmediateStop THEN
				ImmediateStopRequest := TRUE;
				OldState			 := State;
				Feeder_ImmediateStop := TRUE;
				Crane_ImmediateStop  := TRUE;
				Pallet_ImmediateStop := TRUE;
				State				 := M_StopSequence;
			END_IF;

			IF OnPhaseStop THEN
				OnPhaseStopRequest := TRUE;
				OldState		   := State;
				Feeder_OnPhaseStop := TRUE;
				Crane_OnPhaseStop  := TRUE;
				Pallet_OnPhaseStop := TRUE;
				State			   := M_StopSequence;
			END_IF;

		// Pallet is reaching the correct position in order to load the boxes and the cartboard on it

		M_WaitForPallet:

			IF PalletReady THEN
				BoxesOnCrane	  := FALSE;
				LoadBoxesOnPallet := TRUE;
				State			  := M_BoxOnPallet;
			END_IF;

			IF EmergencyStop THEN
				Feeder_EmergencyStop := TRUE;
				Crane_EmergencyStop  := TRUE;
				Pallet_EmergencyStop := TRUE;
				State				 := M_EmergencyStopSequence;
			END_IF;

			IF ImmediateStop THEN
				ImmediateStopRequest := TRUE;
				OldState			 := State;
				Feeder_ImmediateStop := TRUE;
				Crane_ImmediateStop  := TRUE;
				Pallet_ImmediateStop := TRUE;
				State				 := M_StopSequence;
			END_IF;

			IF OnPhaseStop THEN
				OnPhaseStopRequest := TRUE;
				OldState		   := State;
				Feeder_OnPhaseStop := TRUE;
				Crane_OnPhaseStop  := TRUE;
				Pallet_OnPhaseStop := TRUE;
				State			   := M_StopSequence;
			END_IF;

		// Both layers of boxer and  both cartboards are placed on the pallet

		M_BoxOnPallet:

			IF BoxesOnPallet THEN
				HoldBoxes		  := FALSE;
				LoadBoxesOnPallet := FALSE;

				IF SecondLayer THEN
					PalletExit_EN	:= TRUE;
					State			:= M_PalletExit;
				END_IF;

				IF NOT SecondLayer THEN
					State := M_WaitStart;
				END_IF;
			END_IF;

			IF EmergencyStop THEN
				Feeder_EmergencyStop := TRUE;
				Crane_EmergencyStop  := TRUE;
				Pallet_EmergencyStop := TRUE;
				State				 := M_EmergencyStopSequence;
			END_IF;

			IF ImmediateStop THEN
				ImmediateStopRequest := TRUE;
				OldState			 := State;
				Feeder_ImmediateStop := TRUE;
				Crane_ImmediateStop  := TRUE;
				Pallet_ImmediateStop := TRUE;
				State				 := M_StopSequence;
			END_IF;

			IF OnPhaseStop THEN
				OnPhaseStopRequest := TRUE;
				OldState		   := State;
				Feeder_OnPhaseStop := TRUE;
				Crane_OnPhaseStop  := TRUE;
				Pallet_OnPhaseStop := TRUE;
				State			   := M_StopSequence;
			END_IF;

		// Pallet is ready to leave the station

		M_PalletExit:

			IF PalletExit_DONE THEN
				PalletReady	    := FALSE;
				PalletExit_EN	:= FALSE;
				SecondLayer		:= FALSE;
				PalletOutput 	:= PalletOutput + 1;
				State			:= M_WaitStart;
			END_IF;

			IF EmergencyStop THEN
				Feeder_EmergencyStop := TRUE;
				Crane_EmergencyStop  := TRUE;
				Pallet_EmergencyStop := TRUE;
				State				 := M_EmergencyStopSequence;
			END_IF;

			IF ImmediateStop THEN
				ImmediateStopRequest := TRUE;
				OldState			 := State;
				Feeder_ImmediateStop := TRUE;
				Crane_ImmediateStop  := TRUE;
				Pallet_ImmediateStop := TRUE;
				State				 := M_StopSequence;
			END_IF;

			IF OnPhaseStop THEN
				OnPhaseStopRequest := TRUE;
				OldState		   := State;
				Feeder_OnPhaseStop := TRUE;
				Crane_OnPhaseStop  := TRUE;
				Pallet_OnPhaseStop := TRUE;
				State			   := M_StopSequence;
			END_IF;

	END_CASE;

END_PROGRAM
```

### Program Logical/SignalManager (IEC)

#### SignalMng.st - Cyclic code
```iecst
PROGRAM _CYCLIC

	IF (OperationType = Init) THEN
		SignalManagement (OperationType := Init);
		SignalManagement (OperationType := StartConfiguration);
		SignalManagement.OperationType  := Configuration;
		OperationType 					:= Run;
	ELSE
		SignalManagement (OperationType := StartGeneration);
		SignalManagement.OperationType  := Generation;
	END_IF;

	SignalManagement
	(SignalType  	 := Alarm,
	SignalCode   	 := mOnPhaseStopRequested,
	SignalOutput 	 := OnPhaseStopSIG,
	ActivationSignal := OnPhaseStopButton,
	);

	SignalManagement
	(SignalType 	 := Alarm OR AuxReset,
	SignalCode 		 := mEmergencyStopRequested,
	SignalOutput 	 := EmergencyStopSIG,
	ActivationSignal := EmergencyStopButton,
	);

	(*** FEEDER GROUP FAULTS	***)

	(* Conveyor if fault *)
	SignalManagement
	(SignalType 	 := Alarm OR AuxReset,
	SignalCode		 := mConveyorIfFault,
	SignalOutput 	 := ImmediateStopSIG,
	ActivationSignal := act_ConveyorIFFault,
	);

	(* Pusher fault *)
	SignalManagement
	(SignalType 	 := Alarm OR AuxReset,
	SignalCode 		 := mFeederPusherFault,
	SignalOutput 	 := ImmediateStopSIG,
	ActivationSignal := act_FeederPusherFault,
	);

	(* conveyor turn 1 fault *)
	SignalManagement
	(SignalType 	 := Alarm OR AuxReset,
	SignalCode 		 := mConveyorTurn1Fault,
	SignalOutput 	 := ImmediateStopSIG,
	ActivationSignal := act_ConveyorTurn1Fault,
	);

	(* Turnpusher fault *)
	SignalManagement
	(SignalType 	 := Alarm OR AuxReset,
	SignalCode 		 := mTurnpusherFault,
	SignalOutput 	 := ImmediateStopSIG,
	ActivationSignal := act_TurnpusherFault,
	);

	(* conveyor end fault *)
	SignalManagement
	(SignalType 	 := Alarm OR AuxReset,
	SignalCode 	 	 := mConveyorEndFault,
	SignalOutput 	 := ImmediateStopSIG,
	ActivationSignal := act_ConveyorEndFault,
	);

	(* Carriage fault *)
	SignalManagement
	(SignalType 	 := Alarm OR AuxReset,
	SignalCode 		 := mCarriageFault,
	SignalOutput 	 := ImmediateStopSIG,
	ActivationSignal := act_CarriageFault,
	);

	(*** CRANE GROUP FAULTS ***)

	(* Box crane fault *)
	SignalManagement
	(SignalType 	 := Alarm OR AuxReset,
	SignalCode 		 := mBoxCraneFault,
	SignalOutput 	 := ImmediateStopSIG,
	ActivationSignal := act_BoxCraneFault,
	);

	(* Gantry crane fault *)
	SignalManagement
	(SignalType 	 := Alarm OR AuxReset,
	SignalCode 	 	 := mGantryCraneFault,
	SignalOutput 	 := ImmediateStopSIG,
	ActivationSignal := act_GantryCraneFault,
	);

	(* vacuum fault *)
	SignalManagement
	(SignalType 	 := Alarm OR AuxReset,
	SignalCode 		 := mVacuumFault,
	SignalOutput 	 := ImmediateStopSIG,
	ActivationSignal := act_VacuumFault,
	);

	(* cartboard fault *)
	SignalManagement
	(SignalType 	 := Alarm OR AuxReset,
	SignalCode 		 := mCartboardFault,
	SignalOutput 	 := ImmediateStopSIG,
	ActivationSignal := act_CartboardFault
	);

	(* Pusher X fault *)
	SignalManagement
	(SignalType		 := Alarm OR AuxReset,
	SignalCode 		 := mCranePusherxfault,
	SignalOutput 	 := ImmediateStopSIG,
	ActivationSignal := act_PusherXFault,
	);

	(* Pusher Z fault *)
	SignalManagement
	(SignalType 	 := Alarm OR AuxReset,
	SignalCode 		 := mCranePusherzfault,
	SignalOutput 	 := ImmediateStopSIG,
	ActivationSignal := act_PusherZFault,
	);

	(* Slide Rail fault *)
	SignalManagement
	(SignalType 	 := Alarm OR AuxReset,
	SignalCode 	     := mSlideRailFault,
	SignalOutput 	 := ImmediateStopSIG,
	ActivationSignal := act_SlideRailFault,
	);

	(*** PALLET GROUP FAULTS ***)

	(* Lifter fault *)
	SignalManagement
	(SignalType 	 := Alarm OR AuxReset,
	SignalCode 		 := mPalletLifterFault,
	SignalOutput 	 := ImmediateStopSIG,
	ActivationSignal := act_PalletLifterFault,
	);

	(* fork fault *)
	SignalManagement
	(SignalType 	 := Alarm OR AuxReset,
	SignalCode 		 := mPalletforkFault,
	SignalOutput 	 := ImmediateStopSIG,
	ActivationSignal := act_PalletForkFault,
	);

	(* conveyor 1 fault *)
	SignalManagement
	(SignalType 	 := Alarm OR AuxReset,
	SignalCode 	 	 := mPalletConveyor1Fault,
	SignalOutput 	 := ImmediateStopSIG,
	ActivationSignal := act_PalletConveyor1Fault,
	);

	(* conveyor 2 fault *)
	SignalManagement
	(SignalType 	 := Alarm OR AuxReset,
	SignalCode 		 := mPalletConveyor2Fault,
	SignalOutput 	 := ImmediateStopSIG,
	ActivationSignal := act_PalletConveyor2Fault,
	);

	(* PALLET ALMOST OVER Warning *)
	SignalManagement
	(SignalType 	 := Warning,
	SignalCode 		 := mPalletsAlmostOver,
		//	SignalOutput 	 := PalletAlmostOver,
	SignalOutput 	 := MaterialsRunOut,
	ActivationSignal := (PalletCounter = 1),
	);

	(* PALLET OVER Alarm *)
	SignalManagement
	(SignalType 	 := Alarm,
	SignalCode 		 := mPalletsOver,
	SignalOutput 	 := OnPhaseStopSIG,
	ActivationSignal := (PalletCounter = 0),
	);

	(* CARTBOARD ALMOST OVER Warning *)
	SignalManagement
	(SignalType 	 := Warning,
	SignalCode 		 := mCartboardAlmostOver,
		//	SignalOutput	 := CartboardAlmostOver,
	SignalOutput 	 := MaterialsRunOut,
	ActivationSignal := (CraneCartboardCounter = 1),
	);

	(* CARTBOARD OVER Alarm *)
	SignalManagement
	(SignalType 	 := Alarm,
	SignalCode 		 := mCartboardOver,
	SignalOutput 	 := OnPhaseStopSIG,
	ActivationSignal := (CraneCartboardCounter = 0),
	);

	OutputSignals := SignalManagement.SignalOutputs;

	IF (OperationType = RUN) THEN
		SignalManagement (OperationType := RUN); (* outputs selection *)
	END_IF;

	EmergencyStop := ((OutputSignals AND EmergencyStopSIG) = EmergencyStopSIG);

	IF EmergencyStop THEN
		ImmediateStop := FALSE;
		OnPhaseStop	  := FALSE;
	END_IF;

	IF NOT EmergencyStop THEN
		ImmediateStop := ((OutputSignals AND ImmediateStopSIG) = ImmediateStopSIG);
		OnPhaseStop	  := FALSE;
		IF NOT ImmediateStop THEN
			OnPhaseStop := ((OutputSignals AND OnPhaseStopSIG) = OnPhaseStopSIG);
		END_IF;
	END_IF;

	//	OutOfPallet 		:= ((OutputSignals AND PalletAlmostOver) = PalletAlmostOver);
	//	OutOfCartboard		:= ((OutputSignals AND CartboardAlmostOver) = CartboardAlmostOver);

	OnePalletLeft	 	:= (PalletCounter = 1);
	OneCartboardLeft 	:= (CraneCartboardCounter = 1);
	PalletOver	 		:= (PalletCounter = 0);
	CartboardOver 		:= (CraneCartboardCounter = 0);

	IF NOT EmergencyStop AND NOT ImmediateStop AND NOT OnPhaseStop THEN
		OutOfMaterial := ((OutputSignals AND MaterialsRunOut) = MaterialsRunOut);
	ELSE
		OutOfMaterial := FALSE;
	END_IF;

END_PROGRAM
```

#### Variables.var - Local variables
```iecst
VAR CONSTANT
	Init : INT := 0;
	Run : INT := 1;
	StartConfiguration : INT := 2;
	Configuration : INT := 3;
	StartGeneration : INT := 4;
	Generation : INT := 5;
	Alarm : DINT := 2#0000000000000001;
	Warning : DINT := 2#0000000000000011;
	AuxReset : DINT := 2#0000001000000000;
END_VAR
(*Message IDs*)
VAR CONSTANT
	mTurnpusherFault : INT := 1;
	mFeederPusherFault : INT := 2;
	mCranePusherxfault : INT := 3;
	mCranePusherzfault : INT := 4;
	mVacuumFault : INT := 5;
	mPalletforkFault : INT := 6;
	mPalletsOver : INT := 7;
	mCarriageFault : INT := 8;
	mGantryCraneFault : INT := 9;
	mBoxCraneFault : INT := 10;
	mPalletLifterFault : INT := 11;
	mPalletsAlmostOver : INT := 12;
	mOnPhaseStopRequested : INT := 13;
	mEmergencyStopRequested : INT := 14;
	mCartboardAlmostOver : INT := 15;
	mCartboardOver : INT := 16;
	mConveyorIfFault : INT := 17;
	mConveyorTurn1Fault : INT := 18;
	mConveyorEndFault : INT := 19;
	mCartboardFault : INT := 20;
	mSlideRailFault : INT := 21;
	mPalletConveyor1Fault : INT := 22;
	mPalletConveyor2Fault : INT := 23;
END_VAR
(*Output IDs*)
VAR CONSTANT
	EmergencyStopSIG : DWORD := 16#0001;
	ImmediateStopSIG : DWORD := 16#0002;
	OnPhaseStopSIG : DWORD := 16#0004;
	MaterialsRunOut : DWORD := 16#0400;
END_VAR
VAR
	SignalManagement : SignalManager;
	OnPhaseStopButton : BOOL;
	EmergencyStopButton : BOOL;
	OutputSignals : DWORD;
END_VAR
(**)
VAR
	PalletOver : BOOL;
	CartboardOver : BOOL;
	PalletAlmostOver : DWORD := 16#0005;
	CartboardAlmostOver : DWORD := 16#0006;
	OneCartboardLeft : BOOL;
	OnePalletLeft : BOOL;
END_VAR
```

- Visualisation Logical/mappView (not shown)

Listed in the project but not available here: Logical/Global.typ, Logical/Libraries/ComTCP/ComTCP_P/Types.typ, Logical/Libraries/SignalMng/Types.typ, Logical/InputBridge/Types.typ, Logical/InputBridge/Variables.var, Logical/OutputBridge/Types.typ, Logical/OutputBridge/Variables.var, Logical/SignalManager/Types.typ
